(* PLC project Unnamed, Unknown Unnamed 1 *)
(* stored: creationDateTime 2025-10-17T15:19:20, modificationDateTime 2026-02-02T18:29:21 *)

PROGRAM program0
  VAR
    Buzzer AT %QX0.6 : BOOL;
    Fault AT %IX0.2 : BOOL;
    Clear AT %IX0.3 : BOOL;
    Lamp AT %QX0.5 : BOOL := 1;
  END_VAR
  VAR
    Trigger : BOOL;
    TOF0 : TOF;
    TON0 : TON;
    SR0 : SR;
  END_VAR

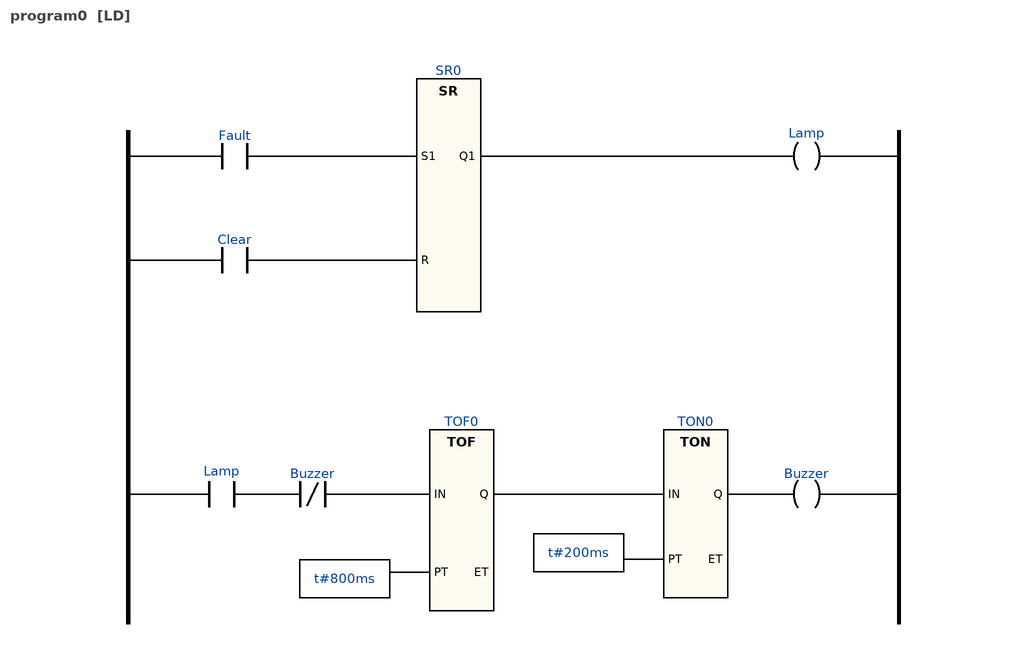
(* LD diagram, written out as Structured Text *)
TOF0(IN := Lamp AND NOT Buzzer, PT := t#800ms);
TON0(IN := TOF0.Q, PT := t#200ms);
Buzzer := TON0.Q;
SR0(S1 := Fault, R := Clear);
Lamp := SR0.Q1;
END_PROGRAM

CONFIGURATION Config0
  RESOURCE Res0 ON PLC
    TASK task0(INTERVAL := T#20ms, PRIORITY := 0);
    PROGRAM instance0 WITH task0 : program0;
  END_RESOURCE
END_CONFIGURATION
